// LS Electric XG5000 project: 1129_LS_DUMP
// PLC NewPLC
// module base 0 slot 0: 입출력 모듈:XBC-DR20S (DC 24V 입력 12점, 릴레이 출력 8점)

PROGRAM dump (task: 스캔 프로그램)

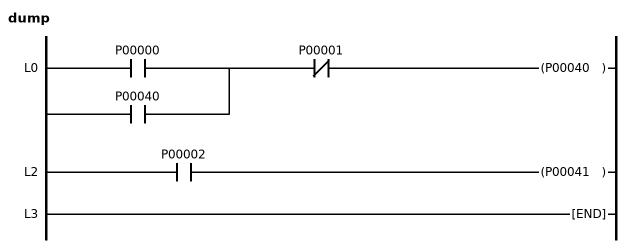
; L0
LOAD      P00000
OR        P00040
AND NOT   P00001
OUT       P00040
; L2
LOAD      P00002
OUT       P00041
; L3
END